PROGRAM P_Mqtt
VAR
  
	sCounter  : STRING(1024);
   
  	// Function blocks for IOT communication 
  	fbMqttClient    : FB_IotMqttClient;
	fbMessageQueue  : FB_IotMqttMessageQueue;
	fbMessage       : FB_IotMqttMessage;	
  
	bSetParameter   : BOOL := TRUE;  // set parametre 
	bHaveNetwork     : BOOL ; 
	
	(* publish message -  *)
	sTopicPub       	: STRING(255);
	sOpStateTopicPub	: STRING(255);
	sPLCStateTopicPub 	: STRING(255);
	sCutStateTopicPub	: STRING(255);
	sPickStateTopicPub	: STRING(255);
	sRecipeTopicPub		: STRING(255);
	sVelocityTopicPub	: STRING(255);
	sProgramTopicPub	: STRING(255);
	
	sPayloadPub     : STRING(255);
	
	bSendMsg         : BOOL;
	
	(* subscription *)
	bSubscribed     : BOOL;
	sTopicSub       : STRING(255);
	
	
	
	(* received message *)
	{attribute 'TcEncoding':='UTF-8'}
	sTopicRcv       : STRING(255);
	{attribute 'TcEncoding':='UTF-8'}
	sPayloadRcv     : STRING(255);
	bError           : BOOL;
	// Sent messages 
	udiSentMessages: UDINT;
	bstatus: BOOL;
	
	fbAdapterInfo: FB_GetAdaptersInfo;
	
	udiCounter : UDINT;
	
	tonSendMsg : Tc2_Standard.TON;
	
	tonMomOn : Tc2_Standard.TON;
	
	sTag : STRING;
	
	iFlag : INT;
	
	bCount : BOOL;
	bForceUpdate : BOOL;
	
END_VAR



 
  A_Init();

  // Connect Action 
  A_Connect();
  
  
  // Send Message Action
  A_SendMessage();
  
  // Subscribe Action
  A_Subscribe();
  
  // Get Adapter Info
  A_AdapterInfo();

ACTION A_AdapterInfo:

fbAdapterInfo(
	sNetID:='' , 
	bExecute:= NOT fbAdapterInfo.bExecute AND NOT fbAdapterInfo.bBusy , 
	tTimeout:= , 
	bBusy=> , 
	bError=> , 
	nErrID=> , 
	arrAdapters=> , 
	nCount=> , 
	nGet=> );
	
IF NOT fbAdapterInfo.bBusy THEN
	IF fbAdapterInfo.arrAdapters[1].sIpAddr <> '0.0.0.0' THEN
		bHaveNetwork:=TRUE;
	ELSE
		bHaveNetwork:=FALSE;
	END_IF
END_IF
END_ACTION

ACTION A_Connect:

// Execute and update MQTT client

fbMqttClient.Execute(bHaveNetwork);
bError:= fbMqttClient.bError;
END_ACTION

ACTION A_Init:

IF bSetParameter THEN

	fbMqttClient.sHostName:='192.168.29.55';
	fbMqttClient.nHostPort:=1883;
	
	fbMqttClient.nKeepAlive := 60;

	fbMqttClient.ipMessageQueue := fbMessageQueue;
		
	bSetParameter  := FALSE;
	
	sTopicPub 			:= 'mqtt/plc2hmi';
	sOpStateTopicPub	:= 'mqtt/plc2hmi/opState';
	sPLCStateTopicPub	:= 'mqtt/plc2hmi/plcState';
	sCutStateTopicPub	:= 'mqtt/plc2hmi/cutState';
	sPickStateTopicPub	:= 'mqtt/plc2hmi/pickState';
	sRecipeTopicPub		:= 'mqtt/plc2hmi/recipe';
	sVelocityTopicPub 	:= 'mqtt/plc2hmi/velocity';
	sProgramTopicPub 	:= 'mqtt/plc2hmi/program';
	
	sTopicSub 			:= 'php-mqtt/hmi2plc/#';
	
ELSIF NOT bHaveNetwork THEN
	bHaveNetwork := FALSE;

END_IF
END_ACTION

ACTION A_SendMessage:
// Send MQTT data 
IF fbMqttClient.bConnected AND bHaveNetwork THEN

	IF PROGRAM_DATA.usiRecipe <> PROGRAM_DATA.usiNewRecipe THEN
		///////////////////////////// RECIPE UPDATE //////////////////////////////
		PROGRAM_DATA.usiRecipe := PROGRAM_DATA.usiNewRecipe;
		sPayloadPub := USINT_TO_STRING(PROGRAM_DATA.usiRecipe);
		bstatus := fbMqttClient.Publish(sTopic:= sRecipeTopicPub, pPayload:= ADR(sPayloadPub), nPayloadSize:= LEN2(ADR(sPayloadPub)), eQoS:= TcIotMqttQos.AtMostOnceDelivery, bRetain:= TRUE, bQueue:= TRUE );
		udiSentMessages := udiSentMessages + 1; 
	END_IF

	IF bPLCStatus <> NewbPLCStatus OR bRobotCutStatus <> NewbRobotCutStatus OR bRobotPickStatus <> NewbRobotPickStatus THEN
		bPLCStatus 			:= NewbPLCStatus;
		bRobotCutStatus		:= NewbRobotCutStatus;
		bRobotPickStatus	:= NewbRobotPickStatus;
		
		// Onchange, publish PLC/Cut/Pick State
		sPayloadPub := BOOL_TO_STRING(bPLCStatus);
		bstatus := fbMqttClient.Publish(sTopic:= sPLCStateTopicPub, pPayload:= ADR(sPayloadPub), nPayloadSize:= LEN2(ADR(sPayloadPub)), eQoS:= TcIotMqttQos.AtMostOnceDelivery, bRetain:= TRUE, bQueue:= TRUE );
		udiSentMessages := udiSentMessages + 1; 
		
		sPayloadPub := BOOL_TO_STRING(bRobotCutStatus);
		bstatus := fbMqttClient.Publish(sTopic:= sCutStateTopicPub, pPayload:= ADR(sPayloadPub), nPayloadSize:= LEN2(ADR(sPayloadPub)), eQoS:= TcIotMqttQos.AtMostOnceDelivery, bRetain:= TRUE, bQueue:= TRUE );
		udiSentMessages := udiSentMessages + 1; 
		
		sPayloadPub := BOOL_TO_STRING(bRobotPickStatus);
		bstatus := fbMqttClient.Publish(sTopic:= sPickStateTopicPub, pPayload:= ADR(sPayloadPub), nPayloadSize:= LEN2(ADR(sPayloadPub)), eQoS:= TcIotMqttQos.AtMostOnceDelivery, bRetain:= TRUE, bQueue:= TRUE );
		udiSentMessages := udiSentMessages + 1; 
	END_IF

	////////////////////////////////// MAIN page HMI ////////////////////////////////////
	IF PROGRAM_DATA.usiProgram <> PROGRAM_DATA.usiNewProgram THEN
		PROGRAM_DATA.usiProgram := PROGRAM_DATA.usiNewProgram;
		
		sPayloadPub := USINT_TO_STRING(PROGRAM_DATA.usiProgram);
		bstatus := fbMqttClient.Publish(sTopic:= sProgramTopicPub, pPayload:= ADR(sPayloadPub), nPayloadSize:= LEN2(ADR(sPayloadPub)), eQoS:= TcIotMqttQos.AtMostOnceDelivery, bRetain:= TRUE, bQueue:= TRUE );
		udiSentMessages := udiSentMessages + 1; 
	END_IF
	
	IF PROGRAM_DATA.usiVelocity <> PROGRAM_DATA.usiNewVelocity THEN
		PROGRAM_DATA.usiVelocity := PROGRAM_DATA.usiNewVelocity;
		
		sPayloadPub := USINT_TO_STRING(PROGRAM_DATA.usiVelocity);
		bstatus := fbMqttClient.Publish(sTopic:= sVelocityTopicPub, pPayload:= ADR(sPayloadPub), nPayloadSize:= LEN2(ADR(sPayloadPub)), eQoS:= TcIotMqttQos.AtMostOnceDelivery, bRetain:= TRUE, bQueue:= TRUE );
		udiSentMessages := udiSentMessages + 1; 
	END_IF
	
	IF bStart AND iFlag <> 1 THEN
		iFlag := 1;
		// When running, publish start
		sPayloadPub := 'start';
		bstatus := fbMqttClient.Publish(sTopic:= sOpStateTopicPub, pPayload:= ADR(sPayloadPub), nPayloadSize:= LEN2(ADR(sPayloadPub)), eQoS:= TcIotMqttQos.AtMostOnceDelivery, bRetain:= TRUE, bQueue:= TRUE );
		udiSentMessages := udiSentMessages + 1; 
	ELSIF (bStop OR NOT bStart) AND iFlag <> 2 THEN
		iFlag := 2;
		// When stopped, publish stop
		sPayloadPub := 'stop';
		bstatus := fbMqttClient.Publish(sTopic:= sOpStateTopicPub, pPayload:= ADR(sPayloadPub), nPayloadSize:= LEN2(ADR(sPayloadPub)), eQoS:= TcIotMqttQos.AtMostOnceDelivery, bRetain:= TRUE, bQueue:= TRUE );
		udiSentMessages := udiSentMessages + 1; 
	END_IF
	


	IF bSendMsg AND iFlag <> 3 THEN // Send data
		iFlag := 3;
		bSendMsg := FALSE;
		 // Publish method - send payload       
		bstatus := fbMqttClient.Publish(sTopic:= sTopicPub, pPayload:= ADR(sCounter), nPayloadSize:= LEN2(ADR(sCounter)), eQoS:= TcIotMqttQos.AtMostOnceDelivery, bRetain:= FALSE, bQueue:= FALSE );
	  udiSentMessages := udiSentMessages + 1; 
 	END_IF
END_IF
END_ACTION

ACTION A_Subscribe:



// Subscribe (modtage) messages with a connection to AZURE is established
IF fbMqttClient.bConnected THEN
  // Subscribe only if not already subscriped
	IF NOT bSubscribed THEN
    // Call of subscribe Method
		bSubscribed := fbMqttClient.Subscribe(sTopic:=sTopicSub, eQoS:=TcIotMqttQos.AtLeastOnceDelivery);
	END_IF
ELSE
	bSubscribed := FALSE;
END_IF




//Get messages with the use of a queue system
IF fbMessageQueue.nQueuedMessages > 0 THEN
	IF fbMessageQueue.Dequeue(fbMessage:=fbMessage) THEN
		fbMessage.GetTopic(pTopic:=ADR(sTopicRcv), nTopicSize:=SIZEOF(sTopicRcv) );
		fbMessage.GetPayload(pPayload:=ADR(sPayloadRcv), nPayloadSize:=SIZEOF(sPayloadRcv), bSetNullTermination:=TRUE);
		
		sTag := MID(STR:= sTopicRcv, LEN:= Tc2_Standard.LEN(sTopicRcv)-12, POS:= 13);		
		
		IF sTopicRcv = 'php-mqtt/hmi2plc/recipe' THEN
			PROGRAM_DATA.usiNewRecipe := STRING_TO_USINT(sPayloadRcv);
			P_SqlSelectRecipe.bRead := TRUE;
		END_IF
		
		IF sTopicRcv = 'php-mqtt/hmi2plc/program' THEN
			PROGRAM_DATA.usiNewProgram := STRING_TO_USINT(sPayloadRcv);
			P_SqlSelectRecipe.bRead := TRUE;
		END_IF
		
		IF sTopicRcv = 'php-mqtt/hmi2plc/setup' THEN
			IF (sPayloadRcv = 'rob-con') THEN
				bRobotConnect 		:= TRUE;
			ELSIF (sPayloadRcv = 'rob-discon') THEN 	
				bRobotDisconnect	:= TRUE;
			ELSIF (sPayloadRcv = 'calib-check') THEN 	
				bCalibCheck 		:= TRUE;
			END_IF
		END_IF
		
		IF sTopicRcv = 'php-mqtt/hmi2plc/calib' THEN
			startCalibCam1 := TRUE;
			sNewCalib := sPayloadRcv;
		END_IF
		
		IF sTopicRcv = 'php-mqtt/hmi2plc/vision' THEN
			usiVisionCmd := STRING_TO_USINT(sPayloadRcv);
		END_IF
		
		IF sTopicRcv = 'php-mqtt/hmi2plc/tool' THEN
			sToolControl := sPayloadRcv;
		END_IF
		
		IF sTopicRcv = 'php-mqtt/hmi2plc/frameUpdate' THEN
			P_SqlSelectFrame.bRead := TRUE;
		END_IF
		
		IF sTopicRcv = 'php-mqtt/hmi2plc/frameUpdate' THEN
			P_SqlSelectFrame.bRead := TRUE;
		END_IF
		
		IF sTopicRcv = 'php-mqtt/hmi2plc/opState' THEN
			IF (sPayloadRcv = 'start') THEN
				bStart	:= TRUE;
				bStop 	:= FALSE;
			ELSIF (sPayloadRcv = 'pause') THEN
				bStop 	:= TRUE;
				bStart	:= FALSE;
			ELSIF (sPayloadRcv = 'stop') THEN
				bStop := TRUE;
				bStart	:= FALSE;
			END_IF
		END_IF
		
		IF	sPayloadRcv = '1' THEN
			IF sTopicRcv = 'php-mqtt/hmi2plc/resetWith' THEN
				bResetButton := TRUE;
			ELSIF sTopicRcv = 'php-mqtt/hmi2plc/resetWithout' THEN
				bResetButton2 := TRUE;
			ELSIF sTopicRcv = 'php-mqtt/hmi2plc/serviceStart' THEN
				bRobotServiceStart := TRUE;
			ELSIF sTopicRcv = 'php-mqtt/hmi2plc/serviceStop' THEN
				bRobotServiceStop := TRUE;
			ELSIF sTopicRcv = 'php-mqtt/hmi2plc/idle' THEN
				bBackToZero := TRUE;
			END_IF
		END_IF
			
		IF sPayloadRcv = '0' THEN
			IF sTopicRcv = 'php-mqtt/hmi2plc/resetWith' THEN
				bResetButton := FALSE;
			ELSIF sTopicRcv = 'php-mqtt/hmi2plc/resetWithout' THEN
				bResetButton2 := FALSE;
			ELSIF sTopicRcv = 'php-mqtt/hmi2plc/serviceStart' THEN
				bRobotServiceStart := FALSE;
			ELSIF sTopicRcv = 'php-mqtt/hmi2plc/serviceStop' THEN
				bRobotServiceStop := FALSE;
			ELSIF sTopicRcv = 'php-mqtt/hmi2plc/idle' THEN
				bBackToZero := FALSE;
			END_IF
			
		END_IF
			
		
		
		IF sTag = 'reset' THEN
			udiCounter := 0;
			bForceUpdate := TRUE;
		ELSIF sTag = 'start' THEN	
			bCount := TO_BOOL(sPayloadRcv);
		END_IF
		
	END_IF
END_IF

tonMomOn(PT:= T#100MS, Q=> , ET=> );
END_ACTION

END_PROGRAM

(* stored: Version 1.1.0.1, ProductVersion 3.1.4024.4
   POU P_Mqtt: Id {1686682f-4c5e-46af-a8e1-7048f3359bbb}, SpecialFunc None
   Action A_AdapterInfo: Id {2e27eef3-6e8d-44b5-986d-a64922301f7a}
   Action A_Connect: Id {51a4e9f4-3b70-4b8a-8a34-378506db0bbd}
   Action A_Init: Id {b75ea88d-e2ae-41cc-a314-9cea5668d546}
   Action A_SendMessage: Id {18bb948d-80b5-4894-8706-11eb4250c15c}
   Action A_Subscribe: Id {1e7a3910-e7c6-48d8-891a-5ba5e0519bf6} *)
